INTERFACE I_SessionStorage

METHOD PUBLIC DisposeSessionDataById
VAR_INPUT
	SessionId : T_MAXSTRING;
	StorageId : T_MAXSTRING;
END_VAR
END_METHOD

METHOD PUBLIC TryRetreiveSessionDataById : BOOL
VAR_INPUT
	SessionId : T_MAXSTRING;
	StorageId : T_MAXSTRING;
	Destination : REFERENCE TO I_SessionData;
END_VAR
END_METHOD

METHOD PUBLIC TryStoreSessionDataById : BOOL
VAR_INPUT
	SessionId : T_MAXSTRING;
	StorageId : T_MAXSTRING;
	Source : I_SessionData;
END_VAR
END_METHOD

END_INTERFACE

(* stored: Version 1.1.0.1, ProductVersion 3.1.4024.12
   Itf I_SessionStorage: Id {45da4111-6767-4006-a93a-ed82aa2a1327}
   Method DisposeSessionDataById: Id {7dc7b73f-f645-486f-8107-5fdea3f2bf35}
   Method TryRetreiveSessionDataById: Id {119bd84a-9a00-4afd-99be-fffb9ae51dfe}
   Method TryStoreSessionDataById: Id {bea07ec3-abca-4cf4-9382-9f53d7172f09} *)
